// TIA Portal V17 export
// export: Created 2024-08-29T18:23:50.1039392Z, ExportSetting WithDefaults, DisplayName Totally Integrated Automation Portal, DisplayVersion V17 Update 7, DisplayName TIA Portal Openness, DisplayVersion V17 Update 7, DisplayName TIA Portal Version Control Interface, DisplayVersion V17, DisplayName SINAMICS Startdrive Advanced, DisplayVersion V17 SP2, DisplayName SINAMICS Startdrive G110M, G120, G120C, G120D, G120P, G115D, DisplayVersion V17 SP2, DisplayName SINAMICS Startdrive G130, G150, S120, S150, SINAMICS MV, S210, DisplayVersion V17 SP2, DisplayName STEP 7 Professional, DisplayVersion V17 Update 7, DisplayName STEP 7 Safety, DisplayVersion V17 Update 6, DisplayName WinCC Advanced / Unified PC, DisplayVersion V17 Update 7
VAR_GLOBAL   // PLC tag table "digitalPLCOutputs"
   qAirInletValve AT %Q0.0 : Bool;
   qLampActivation AT %Q0.4 : Bool;
   qFanActivation AT %Q0.5 : Bool;
   qRedStacklight AT %Q1.7 : Bool;
   qYellowStacklight AT %Q1.6 : Bool;
   qGreenStacklight AT %Q1.5 : Bool;
   qControlIN AT %Q0.6 : Bool;
   qActiveMotor AT %Q0.7 : Bool;
   qDirectionChange AT %Q1.0 : Bool;
   qRedIndicator AT %Q1.1 : Bool;
   qGreenIndicator AT %Q1.2 : Bool;
   qYellowIndicator AT %Q1.3 : Bool;
   qBlueStacklight AT %Q1.4 : Bool;
END_VAR
